FUNCTION_BLOCK ABSTRACT FB_Action EXTENDS FB_OrphanObject IMPLEMENTS I_Action
VAR
END_VAR

METHOD ABSTRACT Execute
VAR_INPUT
    ipObject: I_Object;
END_VAR
END_METHOD

END_FUNCTION_BLOCK

(* stored: Version 1.1.0.1, ProductVersion 3.1.4024.12
   POU FB_Action: Id {9670fb6d-ea6b-06f7-2dd3-159de82debfe}, SpecialFunc None
   Method Execute: Id {62893402-59f6-0f6f-1dfc-91c974ee37aa} *)
